{attribute addProperty BoxType "EL2878-0005-0016"}
{attribute addProperty Id "DiagAT %I*BOOL81"}
{attribute addProperty CRC "1289020322"}
{attribute addProperty SizeInBites "8"}
{attribute addProperty SizeInBytes "1"}
TYPE Diagnostic_4CD4E3A2 :
STRUCT
	{attribute addProperty Name "Diag"}
	Diag AT %I* : BOOL;
END_STRUCT
END_TYPE

(* stored: Version 1.2.0.0, ProductVersion 3.1.4024.9
   DUT Diagnostic_4CD4E3A2: Id {5f89ebe2-66ab-44de-9827-13f2c8bb80aa} *)
